# B&R Automation Studio project Lecture_06_jbl
Automation Studio 4.8.2.72

## Configuration Config1

### Task classes (Cpu.sw)
```
Cyclic#4:
  Opgave2 <- Opgave2.prg
Cyclic#6:
  Blinklys_t <- Blinklys_opg_i_timerne.prg
  Opgave1 <- Opgave1.prg
Binaries: udbdef, FWRules, TCData, sysconf, Role, User, iomap, ashwd, asfw, arconfig, ashwac
Libraries: standard, runtime, astime, asieccon
```

## Logical view

### Program Logical/Blinklys_opg_i_timerne

#### Main.st
```iecst
PROGRAM _INIT
	(* Insert code here *)

END_PROGRAM

PROGRAM _CYCLIC
	(* Insert code here *)
	timer(IN := NOT timer.Q, PT := T#1s);
	// Ovenstånde udtryk kan også skrives som følgende, men er mindre smart
	// timer.IN := NOT timer.Q;
	// timer.PT := T#1s;
	// timer();

	IF timer.Q THEN
		light := NOT light;
	END_IF

END_PROGRAM

PROGRAM _EXIT
	(* Insert code here *)

END_PROGRAM
```

### Program Logical/Opgave1

#### Variables.var
```iecst
VAR
	var : USINT;
END_VAR
```

#### Main.st
```iecst
PROGRAM _INIT
	(* Insert code here *)

END_PROGRAM

PROGRAM _CYCLIC
	(* Insert code here *)

	var := var + 1;

END_PROGRAM

PROGRAM _EXIT
	(* Insert code here *)

END_PROGRAM
```

### Program Logical/Opgave2

#### Variables.var
```iecst
VAR
	shift : BOOL;
	lights : ARRAY[0..15] OF BOOL;
	tmp : BOOL;
END_VAR
```

#### Main.st
```iecst
PROGRAM _INIT
	(* Insert code here *)

	lights[0] := TRUE;

END_PROGRAM

PROGRAM _CYCLIC
	(* Insert code here *)

	IF (shift) THEN
		tmp := lights[0];
		lights[0] := lights[1];
		lights[1] := lights[2];
		lights[2] := lights[3];
		lights[3] := lights[4];
		lights[4] := lights[5];
		lights[5] := lights[6];
		lights[6] := lights[7];
		lights[7] := lights[8];
		lights[8] := lights[9];
		lights[9] := lights[10];
		lights[10] := lights[11];
		lights[11] := lights[12];
		lights[12] := lights[13];
		lights[13] := lights[14];
		lights[14] := lights[15];
		lights[15] := tmp;
	END_IF

END_PROGRAM

PROGRAM _EXIT
	(* Insert code here *)

END_PROGRAM
```
